INTERFACE I_NodeExecuteEndEvent EXTENDS I_Event

PROPERTY PUBLIC CpuCounterHighBytes : UDINT
GET
END_GET
END_PROPERTY

PROPERTY PUBLIC CpuCounterLowBytes : UDINT
GET
END_GET
END_PROPERTY

PROPERTY PUBLIC Target : I_Node
GET
END_GET
END_PROPERTY

END_INTERFACE

(* stored: Version 1.1.0.1, ProductVersion 3.1.4024.13
   Itf I_NodeExecuteEndEvent: Id {2e85dd43-4463-4c45-aae0-9bd8f223fe4e}
   Property CpuCounterHighBytes: Id {b1179647-0966-03b1-1d04-2df626491413}
   Get Get: Id {5aee0dad-0ceb-0412-15ae-c9e2fb2de15b}
   Property CpuCounterLowBytes: Id {64a02129-d2cf-0053-067e-a2551997bb98}
   Get Get: Id {9b87d76c-46cd-0cb1-0f0f-967154155ec0}
   Property Target: Id {ec3f884e-0ea0-43c3-96f1-19fb0f3723e1}
   Get Get: Id {6bfbe76f-3f78-46bd-8222-a68d733fb8ff} *)
